INTERFACE I_CalcXRayAbsorptionConstant EXTENDS I_Fallible


METHOD Calculate
VAR_INPUT
    MaterialFormula : T_MaxString;
    AbsorptionConstant : I_QuantityLREALPublic;
END_VAR
END_METHOD

END_INTERFACE

(* stored: Version 1.1.0.1
   Itf I_CalcXRayAbsorptionConstant: Id {32dae885-22cf-446e-b894-15ca89e88ae3}
   Method Calculate: Id {7fa6b733-5951-4662-96fc-0668fb6204b3} *)
